// TwinCAT 3 PLC project PLC
// Title: Test
// Company: Gema
// Author: RG
// ProjectVersion: 0.1.0.0
// ProgramVersion: 3.1.4023.0
// libraries:
//   Rfid Reader, * (Gema)
//   Tc2_Standard, * (Beckhoff Automation GmbH)
//   Tc2_System, * (Beckhoff Automation GmbH)
//   Tc3_Module, * (Beckhoff Automation GmbH)
//   TcoCore, 0.11.0.2 (Vortex.Library)
//   TcoData, 0.11.0.2 (Vortex.Library)
//   TcoDrivesBeckhoff, 0.11.0.2 (Vortex.Library)
//   TcoElements, 0.11.0.2 (Vortex.Library)
//   TcoPneumatics, 0.11.0.2 (Vortex.Library)
// project tree:
//   / PlcTask.TcTTO (not stored)
//   POUs/ AppContext.TcPOU (not stored), MAIN.TcPOU (not stored), MainStation.TcPOU
// real-time tasks:
//   TASK PlcTask: cycle T#1ms, priority 20, ADS port 350
// I/O:
//   DEVICE Device 2 (EtherCAT)
// variable links:
//   PLC/PLC Instance <-> Device 2 (EtherCAT)/Box 1 (TBEC-LL-4RFID-8DXP)
//     PlcTask Inputs/MAIN._app._mainStation.compactRfid.abyRxDataMapCompactMode <-> Module 2 (128 Byte read)/Inputs 128 Byte read/RD
//     PlcTask Inputs/MAIN._app._mainStation.compactRfid.stCompactModeInputMap <-> Module 1 (HF compact)/Inputs HF compact/Resp
//     PlcTask Outputs/MAIN._app._mainStation.compactRfid.abyTxDataMapCompactMode <-> Module 3 (128 Byte write)/Outputs 128 Byte write/WD
//     PlcTask Outputs/MAIN._app._mainStation.compactRfid.stCompactModeOutputMap <-> Module 1 (HF compact)/Outputs HF compact/Cmd

// ---- POUs/MainStation.TcPOU
FUNCTION_BLOCK MainStation EXTENDS TcoCore.TcoObject
VAR
    counter : INT;
END_VAR

VAR
    compactRfid : RG.Rfid_FB_Compact_Wrapper;
    mockNoRfid : RG.RfidMockNoRfidInRange;
    MockWorking : RG.RfidMockWorking;
    turckRfidHead : RG.RfidHead(THIS^, compactRfid, T#200MS,);
    result : T_MaxString;
    _uid, readData, _reset, _write, _lock : BOOL;

    _isError : BOOL;
    _uiDataRxLength : UINT;
    _uiDataLenght : UINT := 4;

    _errorId : RG.RFID_FB_U.ERROR;

    _offset : byte;
    _data : ARRAY[0..8] OF BYTE := [0, 2, 4, 6];

    _statusLocked : bool;
END_VAR

//counter := counter + 1;

//IF (THIS^.counter MOD 13 = 0) THEN
//    THIS^.Messenger.Info('opalalla').Pin();
//END_IF

//IF (THIS^.counter MOD 400 = 0) THEN
//    THIS^.Messenger.Error('ich Poste').Pin();
//END_IF

turckRfidHead();
_errorId := turckRfidHead.ErrorId;

IF _uid THEN
    IF turckRfidHead.ReadUidMethod().Error THEN
        _isError := turckRfidHead.IsError;
        _errorId := turckRfidHead.ErrorId;
    ELSIF turckRfidHead.ReadUidMethod().Done THEN
        result := turckRfidHead.Uid;
        _uid := FALSE;
    END_IF
END_IF

IF _lock THEN
    _statusLocked := FALSE;
    IF turckRfidHead.LockMethod(1,0).Error THEN
        _isError := turckRfidHead.IsError;
        _errorId := turckRfidHead.ErrorId;
    ELSIF turckRfidHead.LockTask.Done THEN
        _lock := FALSE;
        _statusLocked := TRUE;
    END_IF
END_IF

IF readData THEN
    IF turckRfidHead.ReadDataMethod(_uiDataLenght, _offset).Error THEN
        _isError := turckRfidHead.IsError;
        _errorId := turckRfidHead.ErrorId;
    ELSIF turckRfidHead.ReadDataTask.Done THEN
        _uiDataRxLength := turckRfidHead.DataRxLength;
        readData := FALSE;
        result := turckRfidHead.Data;
    END_IF
END_IF

IF _write THEN
    IF turckRfidHead.WriteDataMethod(_data, _offset).Error THEN
        _isError := turckRfidHead.IsError;
        _errorId := turckRfidHead.ErrorId;
    ELSIF turckRfidHead.WriteDataTask.Done THEN
        _uiDataRxLength := turckRfidHead.DataRxLength;
        _write := FALSE;

    END_IF
END_IF

IF _reset THEN
    _reset := FALSE;
    turckRfidHead.Restore();
END_IF

END_FUNCTION_BLOCK
